// TIA Portal V20 export
TYPE "typeCmControlNode"
// stored: Namespace Unit1.Em3
   STRUCT
      Interlock { ExternalWritable := 'False'} : "Unit1.Em3.typeCmControlNodeInterlock";
   END_STRUCT;
END_TYPE
